// TIA Portal V18 export
// export: Created 2026-06-08T17:01:58.5866458Z, ExportSetting WithDefaults, DisplayName Totally Integrated Automation Portal, DisplayVersion V18, DisplayName TIA Portal Openness, DisplayVersion V18, DisplayName TIA Portal Version Control Interface, DisplayVersion V18, DisplayName STEP 7 Professional, DisplayVersion V18, DisplayName STEP 7 Safety, DisplayVersion V18, DisplayName WinCC Professional, DisplayVersion V18
FUNCTION "M2_I/O" : Void   // FC7, LAD
{ S7_Optimized_Access := 'TRUE' }
VERSION : 0.1
// stored: AutoNumber true, IsIECCheckEnabled false, SetENOAutomatically false, UDAEnableTagReadback false
BEGIN

REGION Network 1
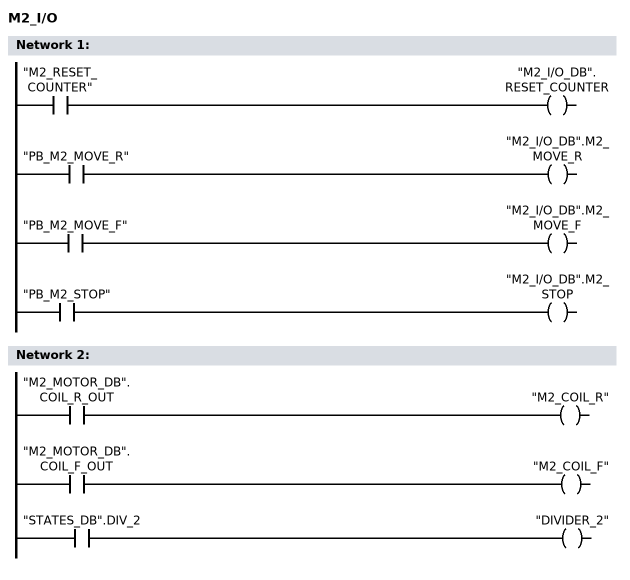
   RUNG wire#powerrail
      Contact( "M2_RESET_COUNTER" )
      Coil( "M2_I/O_DB".RESET_COUNTER )
   END_RUNG
   RUNG wire#powerrail
      Contact( "PB_M2_MOVE_R" )
      Coil( "M2_I/O_DB".M2_MOVE_R )
   END_RUNG
   RUNG wire#powerrail
      Contact( "PB_M2_MOVE_F" )
      Coil( "M2_I/O_DB".M2_MOVE_F )
   END_RUNG
   RUNG wire#powerrail
      Contact( "PB_M2_STOP" )
      Coil( "M2_I/O_DB".M2_STOP )
   END_RUNG
   // the same network as SCL:
   "M2_I/O_DB".RESET_COUNTER := "M2_RESET_COUNTER";
   "M2_I/O_DB".M2_MOVE_R := "PB_M2_MOVE_R";
   "M2_I/O_DB".M2_MOVE_F := "PB_M2_MOVE_F";
   "M2_I/O_DB".M2_STOP := "PB_M2_STOP";
END_REGION

REGION Network 2
   RUNG wire#powerrail
      Contact( "M2_MOTOR_DB".COIL_R_OUT )
      Coil( "M2_COIL_R" )
   END_RUNG
   RUNG wire#powerrail
      Contact( "M2_MOTOR_DB".COIL_F_OUT )
      Coil( "M2_COIL_F" )
   END_RUNG
   RUNG wire#powerrail
      Contact( "STATES_DB".DIV_2 )
      Coil( "DIVIDER_2" )
   END_RUNG
   // the same network as SCL:
   "M2_COIL_R" := "M2_MOTOR_DB".COIL_R_OUT;
   "M2_COIL_F" := "M2_MOTOR_DB".COIL_F_OUT;
   "DIVIDER_2" := "STATES_DB".DIV_2;
END_REGION
END_FUNCTION
